// TIA Portal project "项目1" (V16)

(* hardware
DEVICE "S7-1200 station_1"  S7-1200 Station
   slot 0: "Rack_0"  S7-1200 Rack  Rack  V1.0
   slot 1: "PLC_1"  CPU 1211C DC/DC/DC  6ES7 211-1AE40-0XB0  V4.4
DEVICE "以太网设备_1"  Dummy PC
   slot 1: "PROFINET 接口"  PN-IO
*)

// ===== PLC "PLC_1"  CPU 1211C DC/DC/DC =====

VAR_GLOBAL   // PLC tag table "默认变量表"
   "Tag_1" AT %Q0.0 : Bool;
END_VAR

DATA_BLOCK "DB_ConnPara_1"   // DB1
{ S7_Optimized_Access := 'TRUE' }
VERSION : 0.1
   VAR
      MB_slave : TCON_IP_v4;
   END_VAR
BEGIN
   MB_slave.InterfaceId := 64;
   MB_slave.ID := 16#1;
   MB_slave.ActiveEstablished := 0;
   MB_slave.LocalPort := 502;
END_DATA_BLOCK

DATA_BLOCK "DATA_Slave_1"   // DB2
{ S7_Optimized_Access := 'FALSE' }
VERSION : 0.1
   VAR
      Top1 : Array[1..10] of Int;
      Top2 : Array[1..10] of Int;
   END_VAR
BEGIN
END_DATA_BLOCK

ORGANIZATION_BLOCK "Main"   // OB1, LAD, ProgramCycle
TITLE = "Main Program Sweep (Cycle)"
{ S7_Optimized_Access := 'TRUE' }
VERSION : 0.1
   VAR_INPUT
      Initial_Call : Bool;   // Initial call of this OB
      Remanence : Bool;   // =True, if remanent data are available
   END_VAR
BEGIN

REGION Network 1
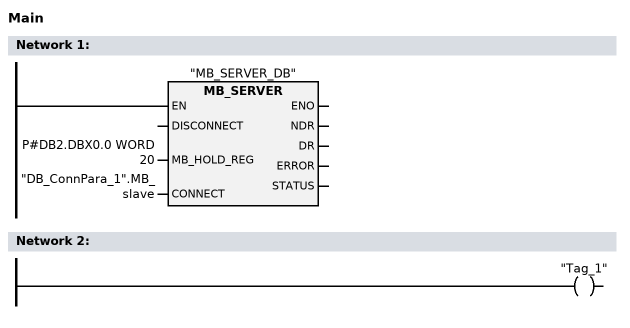
   "MB_SERVER_DB"(MB_HOLD_REG := P#DB2.DBX0.0 WORD 20, CONNECT := "DB_ConnPara_1".MB_slave);   // MB_SERVER
END_REGION

REGION Network 2
   RUNG wire#powerrail
      Coil( "Tag_1" )
   END_RUNG
   // the same network as SCL:
   "Tag_1" := TRUE;
END_REGION
END_ORGANIZATION_BLOCK